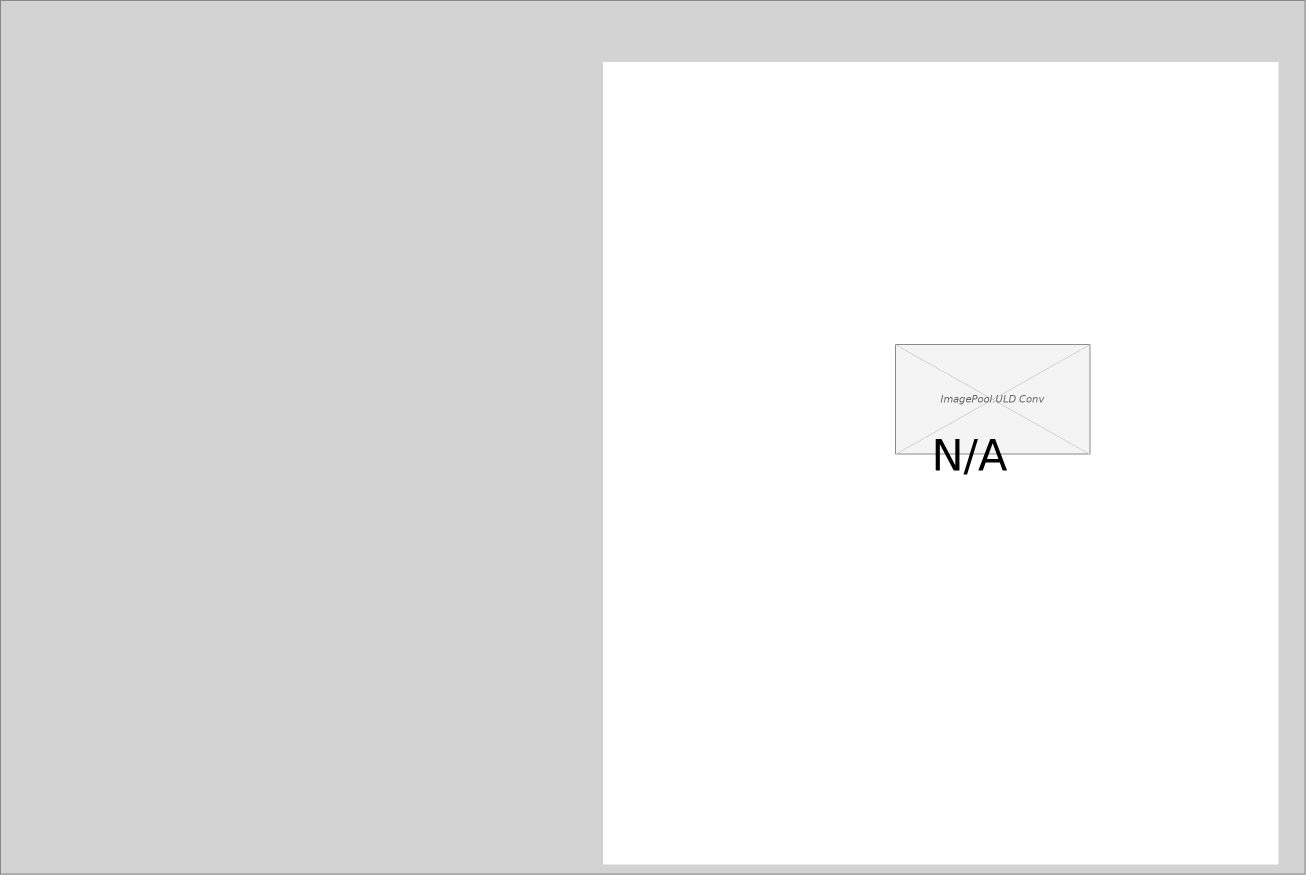
VISUALIZATION Auto_Unloading  // 1306x875
    Rectangle (0,0 1306x875)
    Rectangle (603,62 675x802)
    Image (895,344 195x110), image: ImagePool.ULD Conv
    Label (895,379 149x153), "N/A"
END_VISUALIZATION

(* stored: Version 1.1.0.1, ProductVersion 3.1.4024.12
   Visu Auto_Unloading: Id {ce85721b-66ff-4608-883f-8618f3ed1db2} *)
